{attribute addProperty BoxType "EL1259-0000-0016"}
{attribute addProperty Id "Output_buffer_resetBIT10.1251Manual_output_stateBIT10.1252Force_orderBIT10.1253Output_order_counterUSINT819No_of_output_eventsUSINT8117"}
{attribute addProperty CRC "2881233420"}
{attribute addProperty SizeInBites "67"}
{attribute addProperty SizeInBytes "8.375"}
{warning 'Size of this structure is not a multiple of 8 bits!!!'}
TYPE Ctrl_ABBC220C :
STRUCT
	{attribute addProperty Name "Output_buffer_reset"}
	Output_buffer_reset : BIT;
	{attribute addProperty Name "Manual_output_state"}
	Manual_output_state : BIT;
	{attribute addProperty Name "Force_order"}
	Force_order : BIT;
	{attribute 'hide'}
	reserve_1_BOOL_0 : BOOL;
	{attribute 'hide'}
	reserve_1_BOOL_1 : BOOL;
	{attribute 'hide'}
	reserve_1_BOOL_2 : BOOL;
	{attribute 'hide'}
	reserve_1_BOOL_3 : BOOL;
	{attribute 'hide'}
	reserve_1_BOOL_4 : BOOL;
	{attribute addProperty Name "Output_order_counter"}
	Output_order_counter : USINT;
	{attribute addProperty Name "No_of_output_events"}
	No_of_output_events : USINT;
	{attribute 'hide'}
	reserve_2 : BYTE;
END_STRUCT
END_TYPE

(* stored: Version 1.2.0.0, ProductVersion 3.1.4024.9
   DUT Ctrl_ABBC220C: Id {33bf8a98-e3ca-4ddb-9036-6421fc73b475} *)
